FUNCTION DIJKSTRA
VAR
	i, nMinDistanceNode, nNodeInList, nAdjacentNode, nDistance: INT;
	aVisited : ARRAY[1..24] OF BOOL;
	aParents : ARRAY[1..24] OF INT;
END_VAR

FOR i := 1 TO 24 DO
	GLOBALS.aDistances[i] := CONSTANTS.nIntMax;
	GLOBALS.aRoadFlags[i] := FALSE;
END_FOR

GLOBALS.aDistances[GLOBALS.nStartPosition] := 0;

FOR i := 1 TO 24 DO
	nMinDistanceNode := GET_MIN_DISTANCE_NODE(GLOBALS.aDistances, aVisited);
	aVisited[nMinDistanceNode] := TRUE;
	
	IF NOT (GLOBALS.stGraph.aAdjLists[nMinDistanceNode] = 0) THEN
		FOR nNodeInList := 1 TO 3 DO
			nAdjacentNode := GLOBALS.stGraph.aAdjLists[nMinDistanceNode]^.aAdjNodes[nNodeInList]^.nNode;
			nDistance := GLOBALS.stGraph.aAdjLists[nMinDistanceNode]^.aAdjNodes[nNodeInList]^.nWeight^;
			// z tych 3 warunkow, warunek 2 chyba jest niepotrzebny ale nie pamietam
			IF NOT (aVisited[nAdjacentNode]) AND NOT (GLOBALS.aDistances[nMinDistanceNode] = CONSTANTS.nIntMax) AND (GLOBALS.aDistances[nMinDistanceNode] + nDistance < GLOBALS.aDistances[nAdjacentNode]) THEN
				GLOBALS.aDistances[nAdjacentNode] := GLOBALS.aDistances[nMinDistanceNode] + nDistance;
				aParents[nAdjacentNode] :=  nMinDistanceNode;
			END_IF
		END_FOR
	END_IF
END_FOR

GET_SHORTEST_PATH(GLOBALS.nEndPosition, aParents);

END_FUNCTION

(* stored: Version 1.1.0.1, ProductVersion 3.1.4024.12
   POU DIJKSTRA: Id {f12d046f-06b3-4953-8873-24d60fcc44db}, SpecialFunc None *)
